FUNCTION_BLOCK FB_MyFB2
VAR_INPUT
END_VAR
VAR_OUTPUT
END_VAR
VAR
END_VAR

END_FUNCTION_BLOCK

(* stored: Version 1.1.0.1, ProductVersion 3.1.4024.14
   POU FB_MyFB2: Id {3e9cad39-b7d1-4ec5-a5b4-7870e59d4c5a}, SpecialFunc None *)
